RoboDK station: 001.rdk

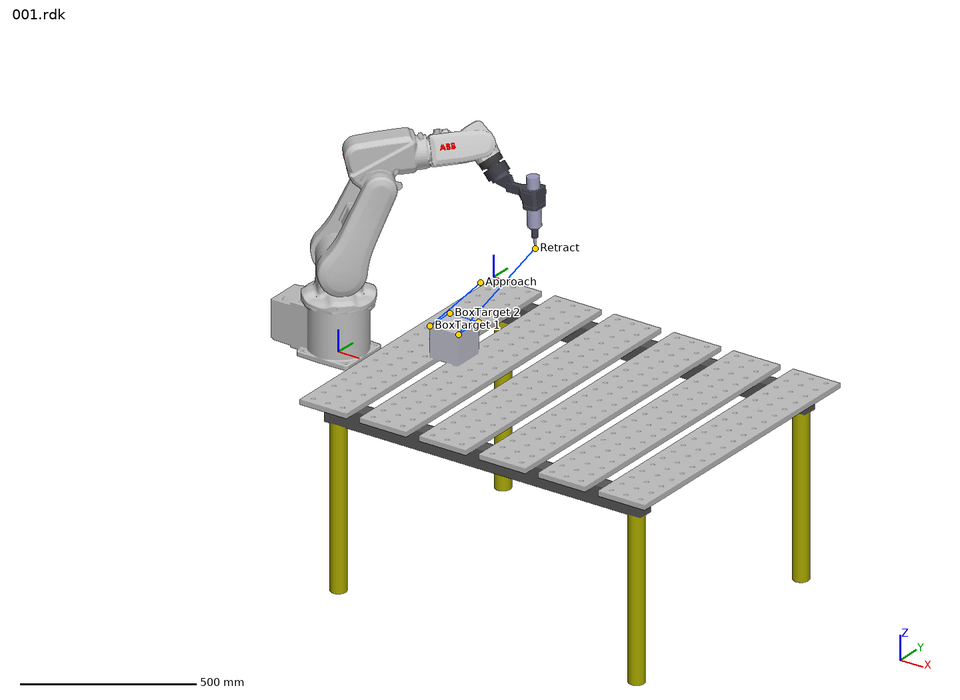
[picture v0: the station drawn from its stored meshes, robots at their saved joint values, targets as dots, program paths as lines]
Station 001 (saved by RoboDK 5.3.4). Poses are relative to the parent item; angles as X-Y-Z fixed-axis rotations.
  - frame ABB IRB 120-3/0.6 Base at (0, 0, 0) mm
    - robot ABB IRB 120-3/0.6: 6 axes, payload 3 kg, reach 580 mm, repeatability 0.01 mm, weight 25 kg
        modified DH rows (alpha deg, a mm, theta deg, d mm): 0, 0, 0, 290; -90, 0, -90, 0; 0, 270, 0, 0; -90, 70, 0, 302; 90, 0, 0, 0; -90, 0, 180, 72
        joint limits [-165, -110, -90, -160, -120, -400] to [165, 110, 70, 160, 120, 400]; home [0, 0, 0, 0, 0, 0]; saved at [41.864, 24.021, -28.503, -28.168, 65.331, 47.067]
      - tool Spindle, TCP at (32, 0, 260) mm, rotated rx 0 ry 39 rz 0 deg, size 157.3 x 72 x 259.9 mm
  - object Table at (800, 0, 100) mm, size 1193.8 x 965.2 x 609.6 mm, geometry from welding_table.sld
  - frame worktable at (200, 480, 100) mm
    - object box at (200, -480, 50) mm, size 100 x 100 x 100 mm, geometry from box.sld
    - target Approach (Cartesian target) at (290.89, -480, 255.1) mm, rotated rx 180 ry 1 rz -180 deg; joints [0, 0, 0, 0, 50, 0] of ABB IRB 120-3/0.6
    - target Retract (Cartesian target) at (290.89, -209.37, 255.1) mm, rotated rx -180 ry 1 rz -180 deg; joints [41.864, 24.021, -28.503, -28.168, 65.331, 47.067] of ABB IRB 120-3/0.6
    - target BoxTarget 1 (Cartesian target) at (152.86, -532.17, 100.05) mm, rotated rx 180 ry 1 rz -180 deg; joints [-17.65, -29.746, 51.98, 22.211, 31.036, -32.981] of ABB IRB 120-3/0.6
    - target BoxTarget 2 (Cartesian target) at (150, -430, 100) mm, rotated rx -180 ry 1 rz -180 deg; joints [17.242, -30.659, 52.497, -21.539, 31.262, 32.017] of ABB IRB 120-3/0.6
    - target BoxTarget 3 (Cartesian target) at (250, -430, 100) mm, rotated rx -180 ry 1 rz -180 deg; joints [10.84, -6.979, 35.579, -18.077, 22.93, 25.077] of ABB IRB 120-3/0.6
    - target BoxTarget 4 (Cartesian target) at (250, -530, 100) mm, rotated rx -180 ry 1 rz -180 deg; joints [-10.84, -6.979, 35.579, 18.077, 22.93, -25.077] of ABB IRB 120-3/0.6
    - object box at (200, -480, 50) mm, size 100 x 100 x 100 mm, geometry from box.sld
  - program Prog1 (6 instructions, listed below)
  - program Main (1 instructions, listed below)
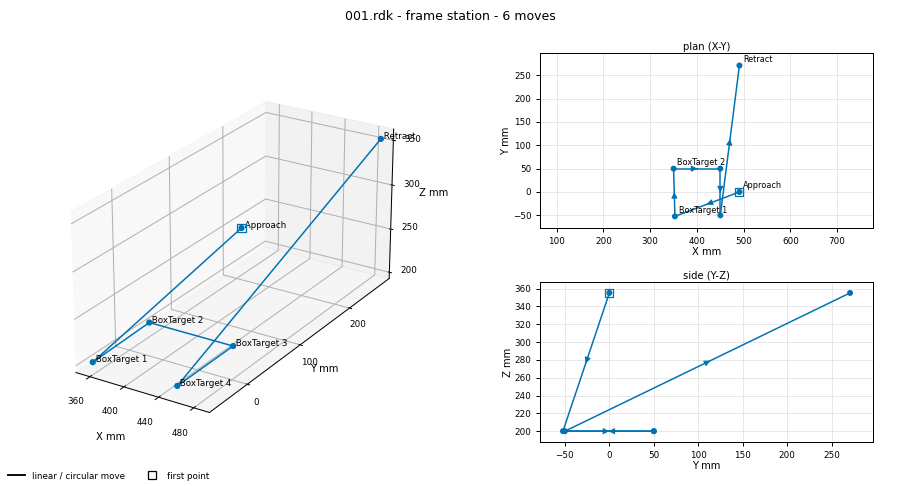
[picture p0: tool path of 001.rdk in frame station, 6 of 6 moves have a stored position in this frame; points joined in program order, loops and branches not executed]

--- program Prog1 (robot ABB IRB 120-3/0.6) ---
  MoveJ (Approach)
  MoveL (BoxTarget 1)
  MoveL (BoxTarget 2)
  MoveL (BoxTarget 3)
  MoveL (BoxTarget 4)
  MoveL (Retract)

--- program Main (robot ABB IRB 120-3/0.6) ---
  调用 Prog1
